{attribute 'qualified_only'}
VAR_GLOBAL
	bStart  			AT %Q* : BOOL;
	bStop  				AT %Q* : BOOL;
	bEnableWinch 		AT %Q* : BOOL;
	bEnableCyl  		AT %Q* : BOOL;
	nWinchOut 			AT %Q* : INT := 19660;
	nCylOut  			AT %Q* : INT := 19660;
END_VAR

(* stored: Version 1.1.0.1, ProductVersion 3.1.4024.11
   GVL IO: Id {a29b5855-7385-475c-a018-933bd981cf9c} *)
